{attribute 'linkalways'} 
{attribute 'no_explicit_call' := 'This FB is a CLASS and must be accessed using methods or properties'}
{attribute 'enable_dynamic_creation'}
FUNCTION_BLOCK Node_F_VN_SetAt_DINT EXTENDS VisionNode
VAR
    nElement : _DINT(0);
    ipContainer : _ITcVnContainer;
    nIndex : _ULINT(0);
    hrPrev : _HRESULT(S_OK);
    hresult : _HRESULT(S_OK);
END_VAR

METHOD PUBLIC  Clone : I_Node
VAR
	pNode : POINTER TO Node_F_VN_SetAt_DINT;
END_VAR
pNode := __NEW(Node_F_VN_SetAt_DINT);
Clone := pNode^;
END_METHOD

METHOD FB_init : BOOL
VAR_INPUT
	bInitRetains : BOOL; // if TRUE, the retain variables are initialized (warm start / cold start)
	bInCopyCode : BOOL;  // if TRUE, the instance afterwards gets moved into the copy code (online change)
END_VAR
AddParameter('nElement', nElement);
AddInput('ipContainer', ipContainer);
AddParameter('nIndex', nIndex);
AddInput('hrPrev', hrPrev);
AddOutput('ipContainer', ipContainer);
AddOutput('hresult',hresult);
END_METHOD

METHOD PROTECTED OnExecute
hresult.Value := F_VN_SetAt_DINT(
    nElement := nElement.Value,
    ipContainer := ipContainer.Value,
    nIndex := nIndex.Value,
    hrPrev:= hrPrev.Value);
END_METHOD

METHOD PUBLIC PreExecutionCheck
VAR_INPUT
	Check : I_PreExecutionChecks;
END_VAR
Check.IsTrue(ipContainer.IsValid, 'ipContainer must be a valid container');
Check.IsTrue(ipContainer.IsType(TC_GLOBAL_CONST_LIST.ContainerType_Vector_DINT), 'ipContainer contains incorrect type');
END_METHOD

END_FUNCTION_BLOCK

(* stored: Version 1.1.0.1, ProductVersion 3.1.4026.13
   POU Node_F_VN_SetAt_DINT: Id {c007e8b5-bffc-4680-957b-ea5912b3271a}, SpecialFunc None
   Folder Constructor: Id {97af9efc-2bfe-45eb-a902-7374b6b8ec10}
   Method Clone: Id {45d90af5-6d1d-4b41-84fd-337a46730edb}
   Method FB_init: Id {ef3dcfff-9917-4dff-a7d1-c0cade2bbf78}
   Method OnExecute: Id {abf5569d-ca2b-479d-8a25-e6c0fcb75620}
   Method PreExecutionCheck: Id {e9dd06c4-1099-427a-bc85-6c0b9d1cbc3e} *)
